% RSLogix 500 project WN16_175291_P_WFI_01_1.RSS, saved by version 8.10.00.24 %
PROJECT "RX72EPIS"    % processor: SLC 500, 1747-L541 %

PROGRAM FILES
  LAD 2   11 rungs
  LAD 3 "table_entr"  31 rungs
  LAD 4 "consigne"  87 rungs
  LAD 5 "communicat"  10 rungs
  LAD 6 "alarmes"  55 rungs
  LAD 7 "programme"  27 rungs
  LAD 8 "pid"  41 rungs
  LAD 9 "affichage"  22 rungs
  LAD 10 "table_sort"  54 rungs
  LAD 29 "IN_TOC"  9 rungs  % TABLE ENTREE/ SOUS-ROUTINE TOC %
  LAD 30 "TOC"  25 rungs  % SOUS-ROUTINE TOC %

DATA FILES
  O0 OUTPUT  6 elements
  I1 INPUT  8 elements
  S2 STATUS  164 elements
  B3 BINARY  18 elements
  T4 TIMER  61 elements
  C5 COUNTER  6 elements
  R6 CONTROL  1 elements
  N7 INTEGER  11 elements
  F8 FLOAT  11 elements
  B9   21 elements
  B10   21 elements
  N11   75 elements
  N12   11 elements
  N13   12 elements
  N14   11 elements
  N15   11 elements
  N16   6 elements
  N17   2 elements
  B18   4 elements
  N19   98 elements
  T20   25 elements
  B21   7 elements
  N24   75 elements
  N25   31 elements
  N27   56 elements
  N28   26 elements
  N30 TOC  30 elements  % Data Files/ Analyseur TOC %
  T31 TOC TIMER  10 elements  % Data Files/ Analyseur TOC %

LADDER 2
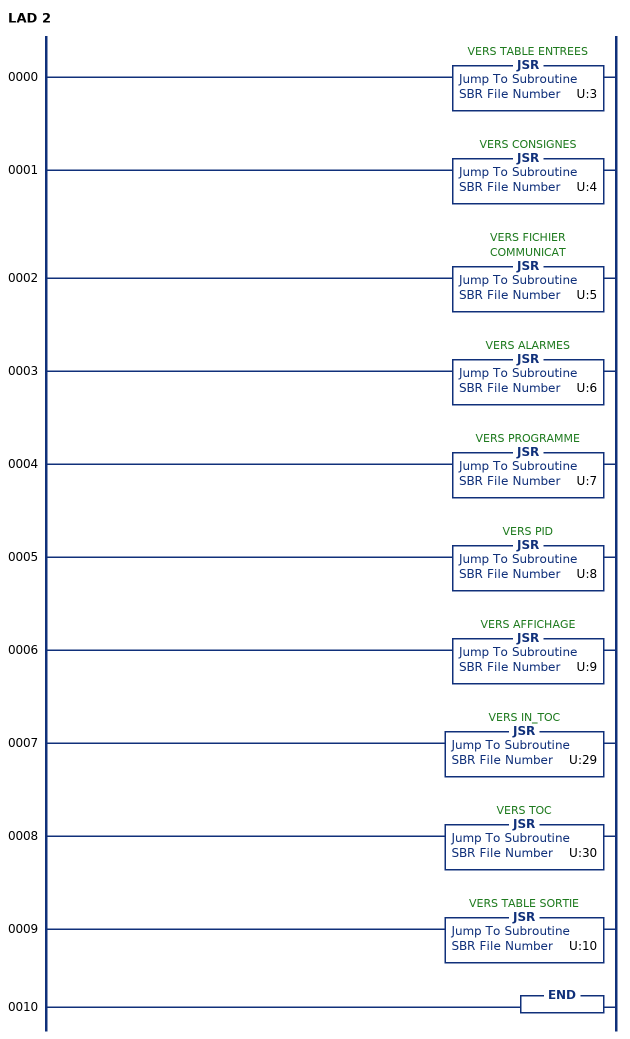
% Rung: 0 %
SOR JSR U:3 EOR
%   U:3  "VERS TABLE ENTREES" %
% Rung: 1 %
SOR JSR U:4 EOR
%   U:4  "VERS CONSIGNES" %
% Rung: 2 %
SOR JSR U:5 EOR
%   U:5  "VERS FICHIER COMMUNICAT" %
% Rung: 3 %
SOR JSR U:6 EOR
%   U:6  "VERS ALARMES" %
% Rung: 4 %
SOR JSR U:7 EOR
%   U:7  "VERS PROGRAMME" %
% Rung: 5 %
SOR JSR U:8 EOR
%   U:8  "VERS PID" %
% Rung: 6 %
SOR JSR U:9 EOR
%   U:9  "VERS AFFICHAGE" %
% Rung: 7 %
SOR JSR U:29 EOR
%   U:29  "VERS IN_TOC" %
% Rung: 8 %
SOR JSR U:30 EOR
%   U:30  "VERS TOC" %
% Rung: 9 %
SOR JSR U:10 EOR
%   U:10  "VERS TABLE SORTIE" %
% Rung: 10 %
SOR END EOR

LADDER 3 "table_entr"
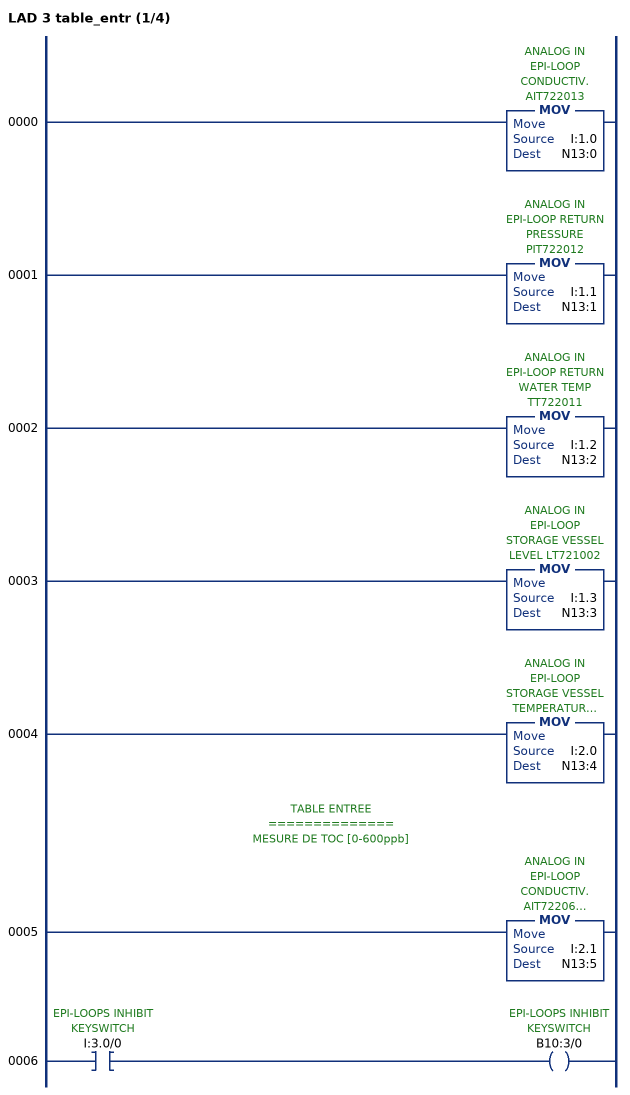
% Rung: 0 %
SOR MOV I:1.0 N13:0 EOR
%   N13:0  "ANALOG IN EPI-LOOP CONDUCTIV. AIT722013" %
% Rung: 1 %
SOR MOV I:1.1 N13:1 EOR
%   N13:1  "ANALOG IN EPI-LOOP RETURN PRESSURE PIT722012" %
% Rung: 2 %
SOR MOV I:1.2 N13:2 EOR
%   N13:2  "ANALOG IN EPI-LOOP RETURN WATER TEMP TT722011" %
% Rung: 3 %
SOR MOV I:1.3 N13:3 EOR
%   N13:3  "ANALOG IN EPI-LOOP STORAGE VESSEL LEVEL LT721002" %
% Rung: 4 %
SOR MOV I:2.0 N13:4 EOR
%   N13:4  "ANALOG IN EPI-LOOP STORAGE VESSEL TEMPERATURE TT721005" %
% Rung: 5 %
% TABLE ENTREE
% ==============
% MESURE DE TOC [0-600ppb] %
SOR MOV I:2.1 N13:5 EOR
%   N13:5  AT_M3  "ANALOG IN EPI-LOOP CONDUCTIV. AIT722062" %
% Rung: 6 %
SOR XIC I:3.0/0 OTE B10:3/0 EOR
%   I:3.0/0  "EPI-LOOPS INHIBIT KEYSWITCH" %
%   B10:3/0  "EPI-LOOPS INHIBIT KEYSWITCH" %

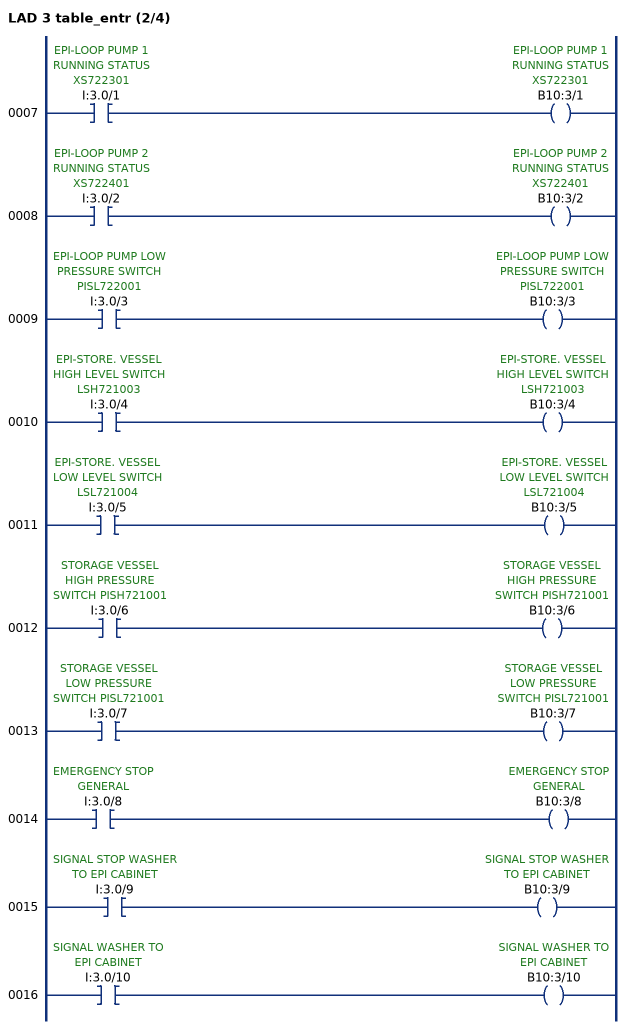
% Rung: 7 %
SOR XIC I:3.0/1 OTE B10:3/1 EOR
%   I:3.0/1  "EPI-LOOP PUMP 1 RUNNING STATUS XS722301" %
%   B10:3/1  "EPI-LOOP PUMP 1 RUNNING STATUS XS722301" %
% Rung: 8 %
SOR XIC I:3.0/2 OTE B10:3/2 EOR
%   I:3.0/2  "EPI-LOOP PUMP 2 RUNNING STATUS XS722401" %
%   B10:3/2  "EPI-LOOP PUMP 2 RUNNING STATUS XS722401" %
% Rung: 9 %
SOR XIC I:3.0/3 OTE B10:3/3 EOR
%   I:3.0/3  "EPI-LOOP PUMP LOW PRESSURE SWITCH PISL722001" %
%   B10:3/3  "EPI-LOOP PUMP LOW PRESSURE SWITCH PISL722001" %
% Rung: 10 %
SOR XIC I:3.0/4 OTE B10:3/4 EOR
%   I:3.0/4  "EPI-STORE. VESSEL HIGH LEVEL SWITCH LSH721003" %
%   B10:3/4  "EPI-STORE. VESSEL HIGH LEVEL SWITCH LSH721003" %
% Rung: 11 %
SOR XIC I:3.0/5 OTE B10:3/5 EOR
%   I:3.0/5  "EPI-STORE. VESSEL LOW LEVEL SWITCH LSL721004" %
%   B10:3/5  "EPI-STORE. VESSEL LOW LEVEL SWITCH LSL721004" %
% Rung: 12 %
SOR XIC I:3.0/6 OTE B10:3/6 EOR
%   I:3.0/6  "STORAGE VESSEL HIGH PRESSURE SWITCH PISH721001" %
%   B10:3/6  "STORAGE VESSEL HIGH PRESSURE SWITCH PISH721001" %
% Rung: 13 %
SOR XIC I:3.0/7 OTE B10:3/7 EOR
%   I:3.0/7  "STORAGE VESSEL LOW PRESSURE SWITCH PISL721001" %
%   B10:3/7  "STORAGE VESSEL LOW PRESSURE SWITCH PISL721001" %
% Rung: 14 %
SOR XIC I:3.0/8 OTE B10:3/8 EOR
%   I:3.0/8  "EMERGENCY STOP GENERAL" %
%   B10:3/8  "EMERGENCY STOP GENERAL" %
% Rung: 15 %
SOR XIC I:3.0/9 OTE B10:3/9 EOR
%   I:3.0/9  "SIGNAL STOP WASHER TO EPI CABINET" %
%   B10:3/9  "SIGNAL STOP WASHER TO EPI CABINET" %
% Rung: 16 %
SOR XIC I:3.0/10 OTE B10:3/10 EOR
%   I:3.0/10  "SIGNAL WASHER TO EPI CABINET" %
%   B10:3/10  "SIGNAL WASHER TO EPI CABINET" %

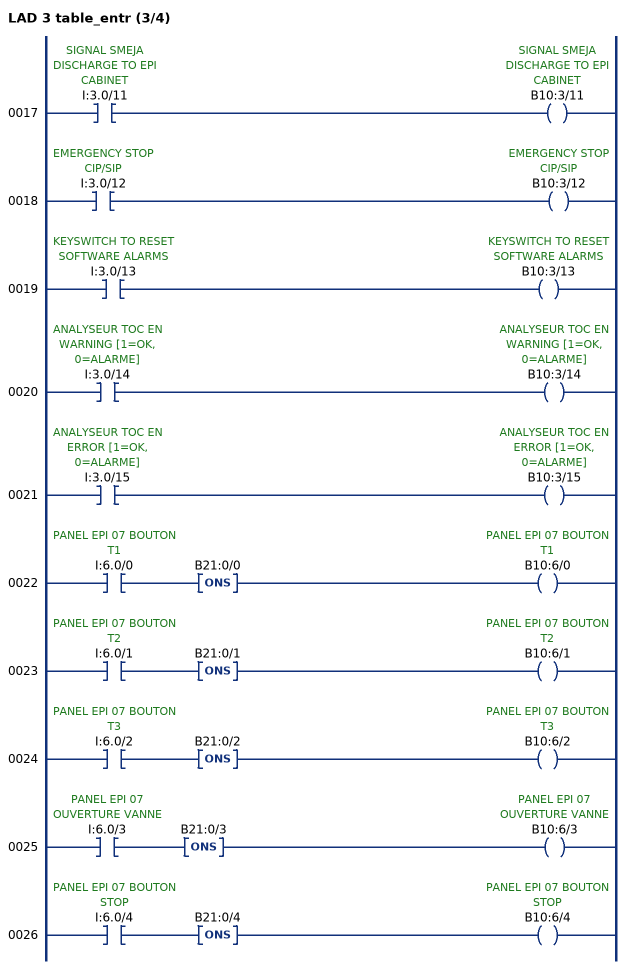
% Rung: 17 %
SOR XIC I:3.0/11 OTE B10:3/11 EOR
%   I:3.0/11  "SIGNAL SMEJA DISCHARGE TO EPI CABINET" %
%   B10:3/11  "SIGNAL SMEJA DISCHARGE TO EPI CABINET" %
% Rung: 18 %
SOR XIC I:3.0/12 OTE B10:3/12 EOR
%   I:3.0/12  "EMERGENCY STOP CIP/SIP" %
%   B10:3/12  "EMERGENCY STOP CIP/SIP" %
% Rung: 19 %
SOR XIC I:3.0/13 OTE B10:3/13 EOR
%   I:3.0/13  "KEYSWITCH TO RESET SOFTWARE ALARMS" %
%   B10:3/13  "KEYSWITCH TO RESET SOFTWARE ALARMS" %
% Rung: 20 %
SOR XIC I:3.0/14 OTE B10:3/14 EOR
%   I:3.0/14  "ANALYSEUR TOC EN WARNING [1=OK, 0=ALARME]" %
%   B10:3/14  "ANALYSEUR TOC EN WARNING [1=OK, 0=ALARME]" %
% Rung: 21 %
SOR XIC I:3.0/15 OTE B10:3/15 EOR
%   I:3.0/15  "ANALYSEUR TOC EN ERROR [1=OK, 0=ALARME]" %
%   B10:3/15  "ANALYSEUR TOC EN ERROR [1=OK, 0=ALARME]" %
% Rung: 22 %
SOR XIC I:6.0/0 OSR B21:0/0 OTE B10:6/0 EOR
%   I:6.0/0  "PANEL EPI 07 BOUTON T1" %
%   B10:6/0  "PANEL EPI 07 BOUTON T1" %
% Rung: 23 %
SOR XIC I:6.0/1 OSR B21:0/1 OTE B10:6/1 EOR
%   I:6.0/1  "PANEL EPI 07 BOUTON T2" %
%   B10:6/1  "PANEL EPI 07 BOUTON T2" %
% Rung: 24 %
SOR XIC I:6.0/2 OSR B21:0/2 OTE B10:6/2 EOR
%   I:6.0/2  "PANEL EPI 07 BOUTON T3" %
%   B10:6/2  "PANEL EPI 07 BOUTON T3" %
% Rung: 25 %
SOR XIC I:6.0/3 OSR B21:0/3 OTE B10:6/3 EOR
%   I:6.0/3  "PANEL EPI 07 OUVERTURE VANNE" %
%   B10:6/3  "PANEL EPI 07 OUVERTURE VANNE" %
% Rung: 26 %
SOR XIC I:6.0/4 OSR B21:0/4 OTE B10:6/4 EOR
%   I:6.0/4  "PANEL EPI 07 BOUTON STOP" %
%   B10:6/4  "PANEL EPI 07 BOUTON STOP" %

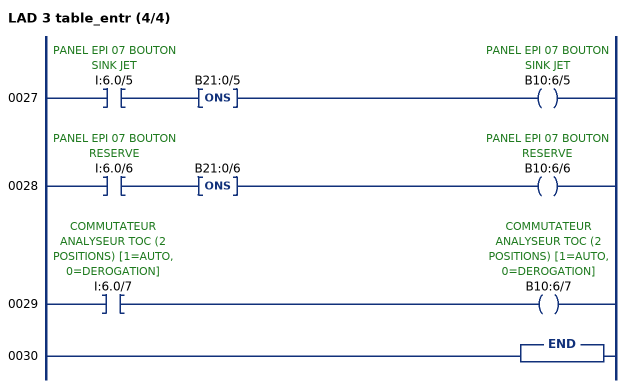
% Rung: 27 %
SOR XIC I:6.0/5 OSR B21:0/5 OTE B10:6/5 EOR
%   I:6.0/5  "PANEL EPI 07 BOUTON SINK JET" %
%   B10:6/5  "PANEL EPI 07 BOUTON SINK JET" %
% Rung: 28 %
SOR XIC I:6.0/6 OSR B21:0/6 OTE B10:6/6 EOR
%   I:6.0/6  "PANEL EPI 07 BOUTON RESERVE" %
%   B10:6/6  "PANEL EPI 07 BOUTON RESERVE" %
% Rung: 29 %
SOR XIC I:6.0/7 OTE B10:6/7 EOR
%   I:6.0/7  "COMMUTATEUR ANALYSEUR TOC (2 POSITIONS) [1=AUTO, 0=DEROGATION]" %
%   B10:6/7  "COMMUTATEUR ANALYSEUR TOC (2 POSITIONS) [1=AUTO, 0=DEROGATION]" %
% Rung: 30 %
SOR END EOR

LADDER 4 "consigne"
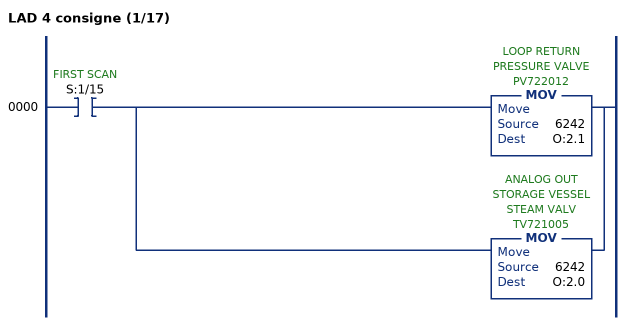
% Rung: 0 %
SOR XIC S:1/15 BST MOV 6242 O:2.1 NXB MOV 6242 O:2.0 BND EOR
%   S:1/15  "FIRST SCAN" %
%   O:2.1  "LOOP RETURN PRESSURE VALVE PV722012" %
%   O:2.0  "ANALOG OUT STORAGE VESSEL STEAM VALV TV721005" %

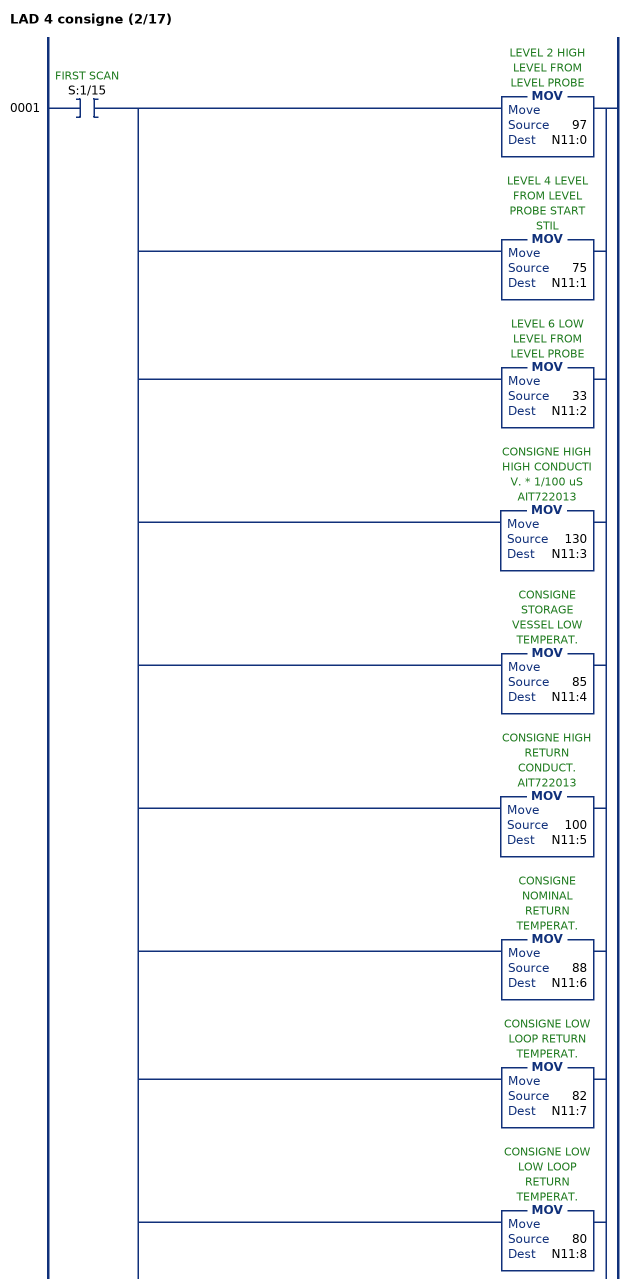

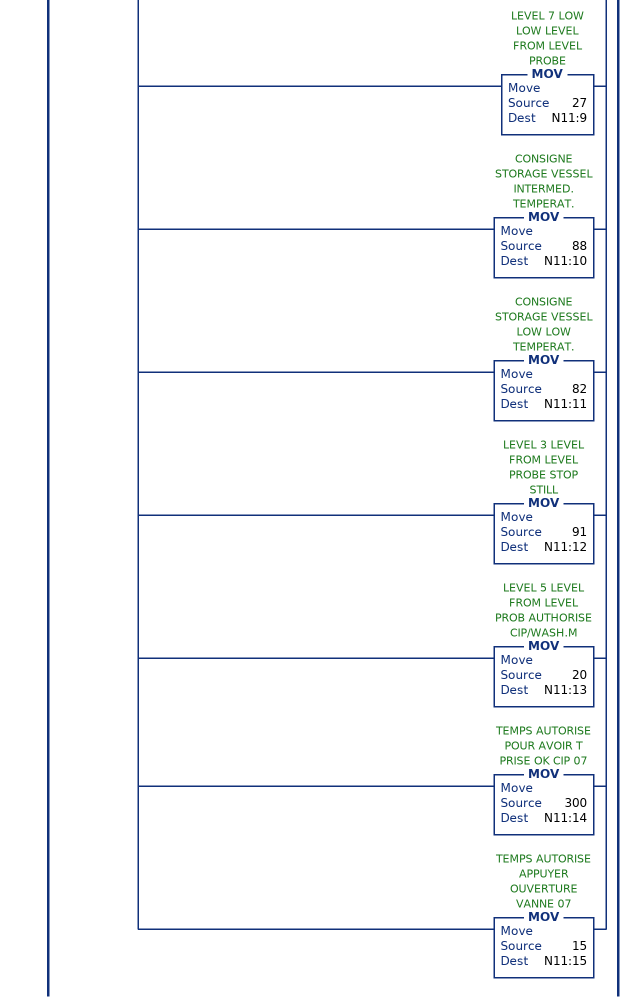
% Rung: 1 %
SOR XIC S:1/15 BST MOV 97 N11:0 NXB MOV 75 N11:1 NXB MOV 33 N11:2 NXB MOV 130 N11:3 NXB MOV 85 N11:4 NXB MOV 100 N11:5 NXB MOV 88 N11:6 NXB MOV 82 N11:7 NXB MOV 80 N11:8 NXB MOV 27 N11:9 NXB MOV 88 N11:10 NXB MOV 82 N11:11 NXB MOV 91 N11:12 NXB MOV 20 N11:13 NXB MOV 300 N11:14 NXB MOV 15 N11:15 BND EOR
%   S:1/15  "FIRST SCAN" %
%   N11:0  "LEVEL 2 HIGH LEVEL FROM LEVEL PROBE" %
%   N11:1  "LEVEL 4 LEVEL FROM LEVEL PROBE START STIL" %
%   N11:2  "LEVEL 6 LOW LEVEL FROM LEVEL PROBE" %
%   N11:3  "CONSIGNE HIGH HIGH CONDUCTIV. * 1/100 uS AIT722013" %
%   N11:4  "CONSIGNE STORAGE VESSEL LOW TEMPERAT." %
%   N11:5  "CONSIGNE HIGH RETURN CONDUCT. AIT722013" %
%   N11:6  "CONSIGNE NOMINAL RETURN TEMPERAT." %
%   N11:7  "CONSIGNE LOW LOOP RETURN TEMPERAT." %
%   N11:8  "CONSIGNE LOW LOW LOOP RETURN TEMPERAT." %
%   N11:9  "LEVEL 7 LOW LOW LEVEL FROM LEVEL PROBE" %
%   N11:10  "CONSIGNE STORAGE VESSEL INTERMED. TEMPERAT." %
%   N11:11  "CONSIGNE STORAGE VESSEL LOW LOW TEMPERAT." %
%   N11:12  "LEVEL 3 LEVEL FROM LEVEL PROBE STOP STILL" %
%   N11:13  "LEVEL 5 LEVEL FROM LEVEL PROB AUTHORISE CIP/WASH.M" %
%   N11:14  "TEMPS AUTORISE POUR AVOIR T PRISE OK CIP 07" %
%   N11:15  "TEMPS AUTORISE APPUYER OUVERTURE VANNE 07" %

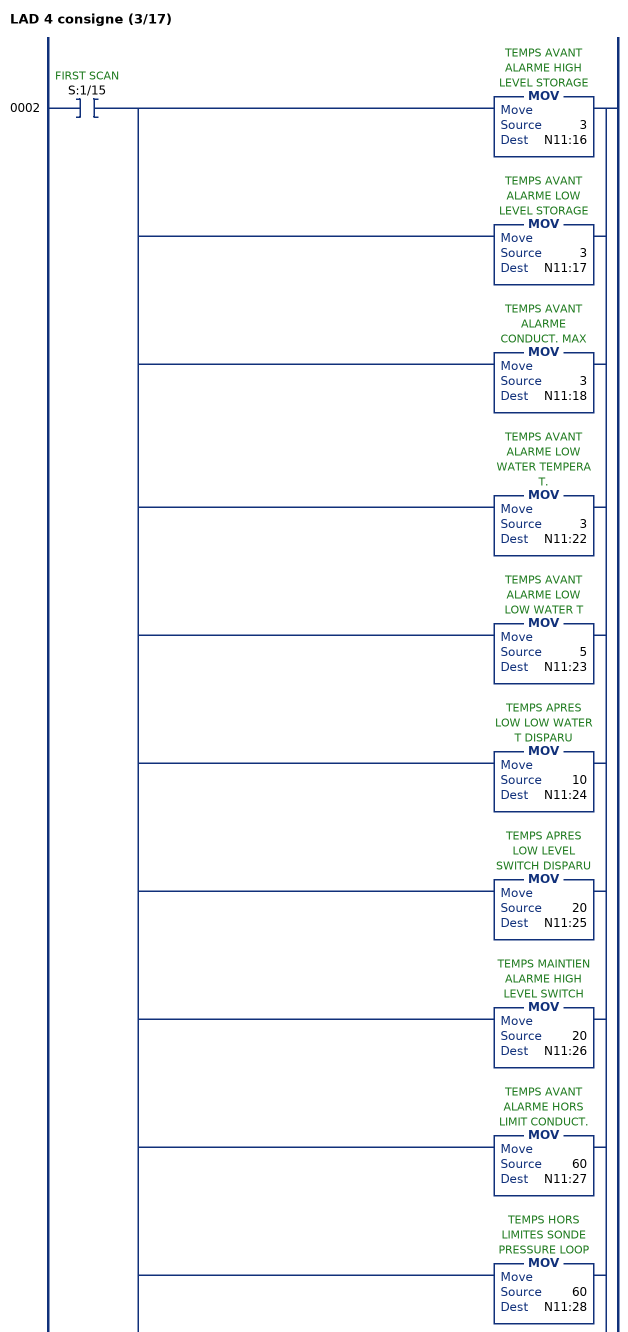

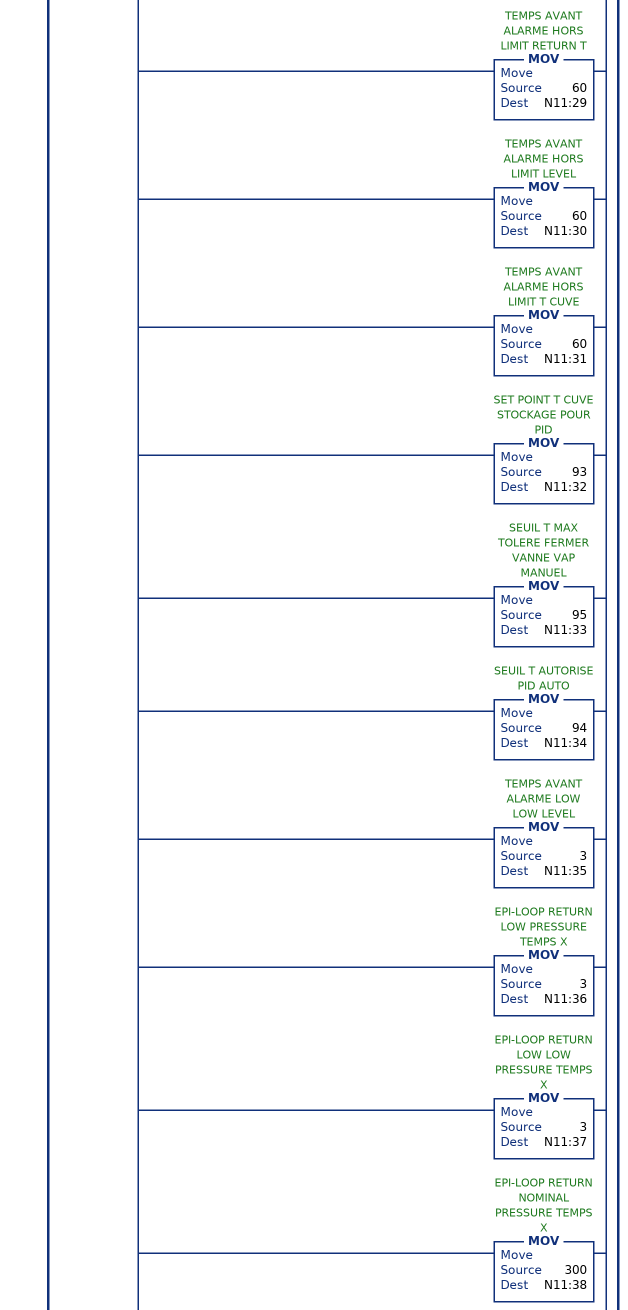

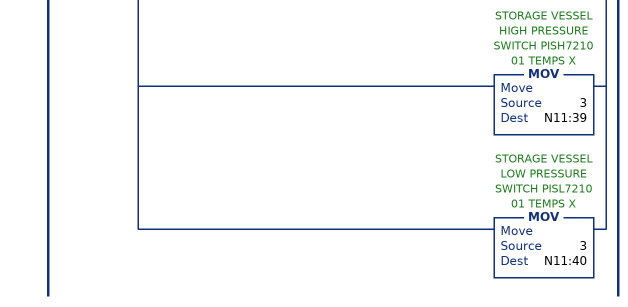
% Rung: 2 %
SOR XIC S:1/15 BST MOV 3 N11:16 NXB MOV 3 N11:17 NXB MOV 3 N11:18 NXB MOV 3 N11:22 NXB MOV 5 N11:23 NXB MOV 10 N11:24 NXB MOV 20 N11:25 NXB MOV 20 N11:26 NXB MOV 60 N11:27 NXB MOV 60 N11:28 NXB MOV 60 N11:29 NXB MOV 60 N11:30 NXB MOV 60 N11:31 NXB MOV 93 N11:32 NXB MOV 95 N11:33 NXB MOV 94 N11:34 NXB MOV 3 N11:35 NXB MOV 3 N11:36 NXB MOV 3 N11:37 NXB MOV 300 N11:38 NXB MOV 3 N11:39 NXB MOV 3 N11:40 BND EOR
%   S:1/15  "FIRST SCAN" %
%   N11:16  "TEMPS AVANT ALARME HIGH LEVEL STORAGE" %
%   N11:17  "TEMPS AVANT ALARME LOW LEVEL STORAGE" %
%   N11:18  "TEMPS AVANT ALARME CONDUCT. MAX" %
%   N11:22  "TEMPS AVANT ALARME LOW WATER TEMPERAT." %
%   N11:23  "TEMPS AVANT ALARME LOW LOW WATER T" %
%   N11:24  "TEMPS APRES LOW LOW WATER T DISPARU" %
%   N11:25  "TEMPS APRES LOW LEVEL SWITCH DISPARU" %
%   N11:26  "TEMPS MAINTIEN ALARME HIGH LEVEL SWITCH" %
%   N11:27  "TEMPS AVANT ALARME HORS LIMIT CONDUCT." %
%   N11:28  "TEMPS HORS LIMITES SONDE PRESSURE LOOP" %
%   N11:29  "TEMPS AVANT ALARME HORS LIMIT RETURN T" %
%   N11:30  "TEMPS AVANT ALARME HORS LIMIT LEVEL" %
%   N11:31  "TEMPS AVANT ALARME HORS LIMIT T CUVE" %
%   N11:32  "SET POINT T CUVE STOCKAGE POUR PID" %
%   N11:33  "SEUIL T MAX TOLERE FERMER VANNE VAP MANUEL" %
%   N11:34  "SEUIL T AUTORISE PID AUTO" %
%   N11:35  "TEMPS AVANT ALARME LOW LOW LEVEL" %
%   N11:36  "EPI-LOOP RETURN LOW PRESSURE TEMPS X" %
%   N11:37  "EPI-LOOP RETURN LOW LOW PRESSURE TEMPS X" %
%   N11:38  "EPI-LOOP RETURN NOMINAL PRESSURE TEMPS X" %
%   N11:39  "STORAGE VESSEL HIGH PRESSURE SWITCH PISH721001 TEMPS X" %
%   N11:40  "STORAGE VESSEL LOW PRESSURE SWITCH PISL721001 TEMPS X" %

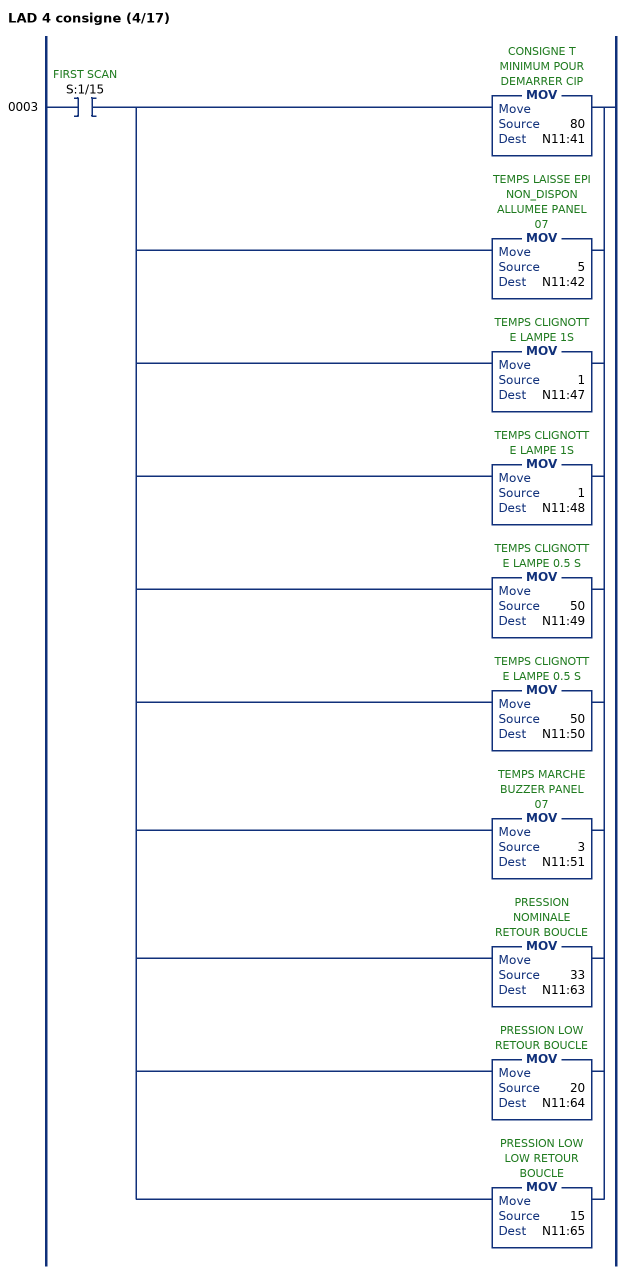
% Rung: 3 %
SOR XIC S:1/15 BST MOV 80 N11:41 NXB MOV 5 N11:42 NXB MOV 1 N11:47 NXB MOV 1 N11:48 NXB MOV 50 N11:49 NXB MOV 50 N11:50 NXB MOV 3 N11:51 NXB MOV 33 N11:63 NXB MOV 20 N11:64 NXB MOV 15 N11:65 BND EOR
%   S:1/15  "FIRST SCAN" %
%   N11:41  "CONSIGNE T MINIMUM POUR DEMARRER CIP" %
%   N11:42  "TEMPS LAISSE EPI NON_DISPON ALLUMEE PANEL 07" %
%   N11:47  "TEMPS CLIGNOTTE LAMPE 1S" %
%   N11:48  "TEMPS CLIGNOTTE LAMPE 1S" %
%   N11:49  "TEMPS CLIGNOTTE LAMPE 0.5 S" %
%   N11:50  "TEMPS CLIGNOTTE LAMPE 0.5 S" %
%   N11:51  "TEMPS MARCHE BUZZER PANEL 07" %
%   N11:63  "PRESSION NOMINALE RETOUR BOUCLE" %
%   N11:64  "PRESSION LOW RETOUR BOUCLE" %
%   N11:65  "PRESSION LOW LOW RETOUR BOUCLE" %

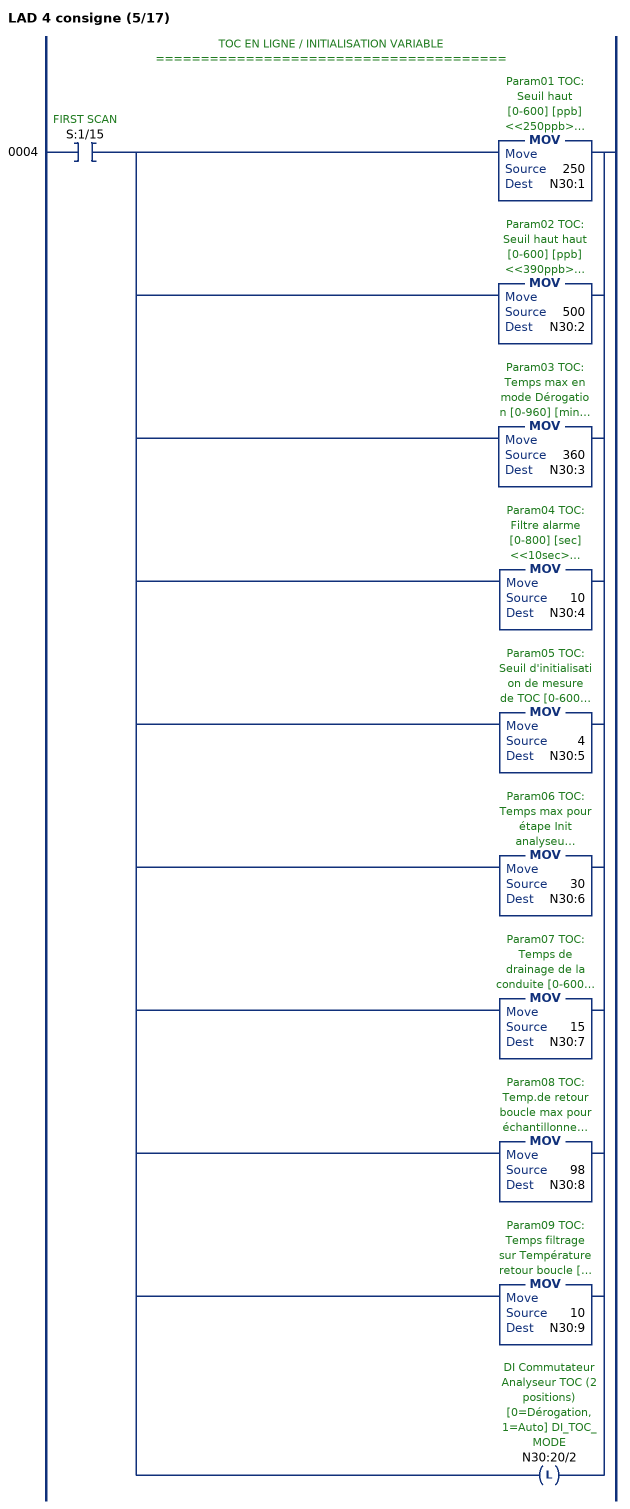
% Rung: 4 %
% TOC EN LIGNE / INITIALISATION VARIABLE
% ======================================= %
SOR XIC S:1/15 BST MOV 250 N30:1 NXB MOV 500 N30:2 NXB MOV 360 N30:3 NXB MOV 10 N30:4 NXB MOV 4 N30:5 NXB MOV 30 N30:6 NXB MOV 15 N30:7 NXB MOV 98 N30:8 NXB MOV 10 N30:9 NXB OTL N30:20/2 BND EOR
%   S:1/15  "FIRST SCAN" %
%   N30:1  AI_AT_M3_LIMH  "Param01 TOC: Seuil haut [0-600] [ppb] <<250ppb>>" %
%   N30:2  AI_AT_M3_LIMHH  "Param02 TOC: Seuil haut haut [0-600] [ppb] <<390ppb>>" %
%   N30:3  AI_TOC_DEROG_LIMH  "Param03 TOC: Temps max en mode Dérogation [0-960] [min] <<360min>>" %
%   N30:4  AI_AT_M3_ALM_HH_DL  "Param04 TOC: Filtre alarme [0-800] [sec] <<10sec>>" %
%   N30:5  AI_AT_M3_MIN  "Param05 TOC: Seuil d'initialisation de mesure de TOC [0-600] [ppb] <<4ppb>>" %
%   N30:6  AI_TOC_INIT_LIMH  "Param06 TOC: Temps max pour étape Init analyseur [0-600] [min] <<30min>>" %
%   N30:7  AI_XV_M3_CMD_DELAY  "Param07 TOC: Temps de drainage de la conduite [0-600] [sec] <<15sec>>" %
%   N30:8  AI_TT_722011_LIMH  "Param08 TOC: Temp.de retour boucle max pour échantillonner [0-100] [°C] <<98°C>>" %
%   N30:9  AI_T_TT_722011_LIMH  "Param09 TOC: Temps filtrage sur Température retour boucle [] [min] <<10 min>>" %
%   N30:20/2  DI_TOC_MODE  "DI Commutateur Analyseur TOC (2 positions) [0=Dérogation, 1=Auto]" %

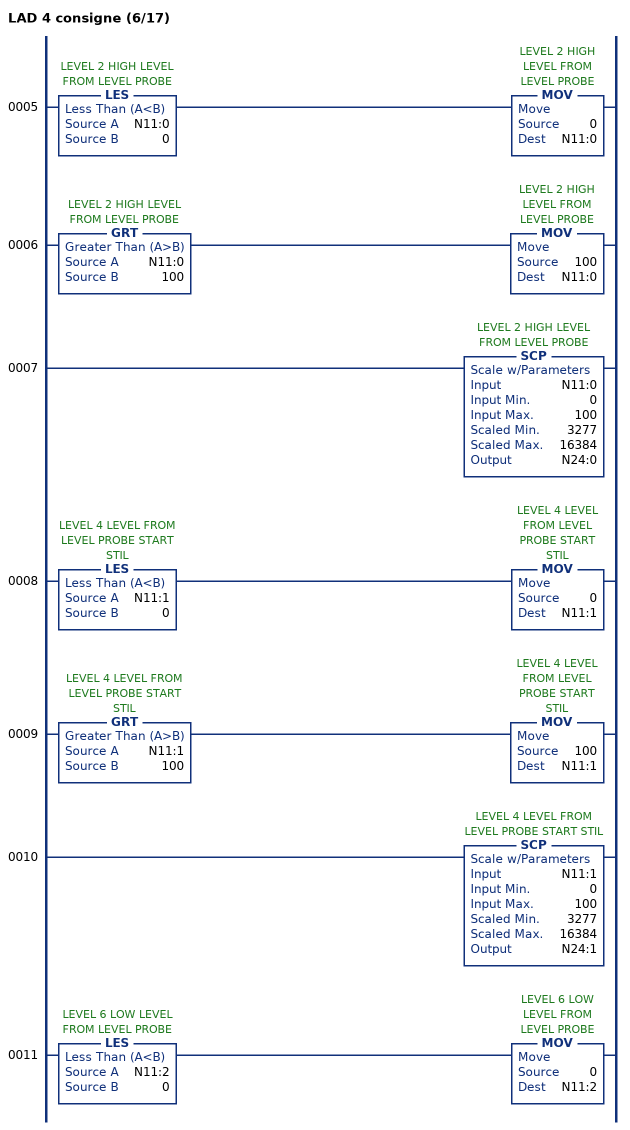
% Rung: 5 %
SOR LES N11:0 0 MOV 0 N11:0 EOR
%   N11:0  "LEVEL 2 HIGH LEVEL FROM LEVEL PROBE" %
% Rung: 6 %
SOR GRT N11:0 100 MOV 100 N11:0 EOR
%   N11:0  "LEVEL 2 HIGH LEVEL FROM LEVEL PROBE" %
% Rung: 7 %
SOR SCP N11:0 0 100 3277 16384 N24:0 EOR
%   N11:0  "LEVEL 2 HIGH LEVEL FROM LEVEL PROBE" %
%   N24:0  "LEVEL 2 HIGH LEVEL FROM LEVEL PROBE" %
% Rung: 8 %
SOR LES N11:1 0 MOV 0 N11:1 EOR
%   N11:1  "LEVEL 4 LEVEL FROM LEVEL PROBE START STIL" %
% Rung: 9 %
SOR GRT N11:1 100 MOV 100 N11:1 EOR
%   N11:1  "LEVEL 4 LEVEL FROM LEVEL PROBE START STIL" %
% Rung: 10 %
SOR SCP N11:1 0 100 3277 16384 N24:1 EOR
%   N11:1  "LEVEL 4 LEVEL FROM LEVEL PROBE START STIL" %
%   N24:1  "LEVEL 4 LEVEL FROM LEVEL PROBE START STIL" %
% Rung: 11 %
SOR LES N11:2 0 MOV 0 N11:2 EOR
%   N11:2  "LEVEL 6 LOW LEVEL FROM LEVEL PROBE" %

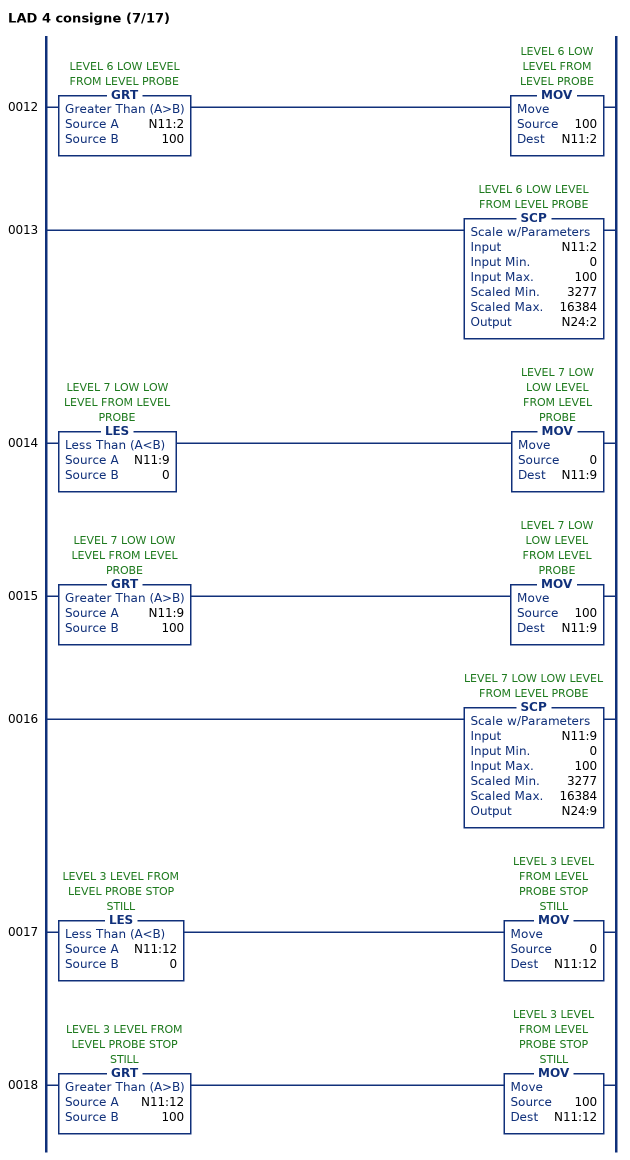
% Rung: 12 %
SOR GRT N11:2 100 MOV 100 N11:2 EOR
%   N11:2  "LEVEL 6 LOW LEVEL FROM LEVEL PROBE" %
% Rung: 13 %
SOR SCP N11:2 0 100 3277 16384 N24:2 EOR
%   N11:2  "LEVEL 6 LOW LEVEL FROM LEVEL PROBE" %
%   N24:2  "LEVEL 6 LOW LEVEL FROM LEVEL PROBE" %
% Rung: 14 %
SOR LES N11:9 0 MOV 0 N11:9 EOR
%   N11:9  "LEVEL 7 LOW LOW LEVEL FROM LEVEL PROBE" %
% Rung: 15 %
SOR GRT N11:9 100 MOV 100 N11:9 EOR
%   N11:9  "LEVEL 7 LOW LOW LEVEL FROM LEVEL PROBE" %
% Rung: 16 %
SOR SCP N11:9 0 100 3277 16384 N24:9 EOR
%   N11:9  "LEVEL 7 LOW LOW LEVEL FROM LEVEL PROBE" %
%   N24:9  "LEVEL 7 LOW LOW LEVEL FROM LEVEL PROBE" %
% Rung: 17 %
SOR LES N11:12 0 MOV 0 N11:12 EOR
%   N11:12  "LEVEL 3 LEVEL FROM LEVEL PROBE STOP STILL" %
% Rung: 18 %
SOR GRT N11:12 100 MOV 100 N11:12 EOR
%   N11:12  "LEVEL 3 LEVEL FROM LEVEL PROBE STOP STILL" %

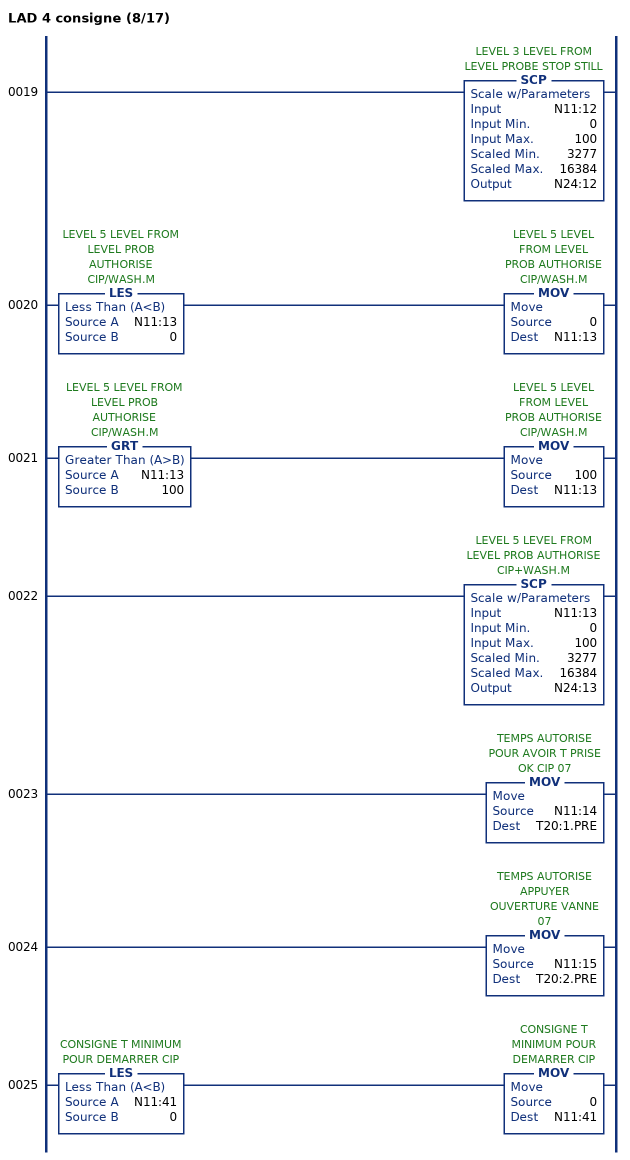
% Rung: 19 %
SOR SCP N11:12 0 100 3277 16384 N24:12 EOR
%   N11:12  "LEVEL 3 LEVEL FROM LEVEL PROBE STOP STILL" %
%   N24:12  "LEVEL 3 LEVEL FROM LEVEL PROBE STOP STILL" %
% Rung: 20 %
SOR LES N11:13 0 MOV 0 N11:13 EOR
%   N11:13  "LEVEL 5 LEVEL FROM LEVEL PROB AUTHORISE CIP/WASH.M" %
% Rung: 21 %
SOR GRT N11:13 100 MOV 100 N11:13 EOR
%   N11:13  "LEVEL 5 LEVEL FROM LEVEL PROB AUTHORISE CIP/WASH.M" %
% Rung: 22 %
SOR SCP N11:13 0 100 3277 16384 N24:13 EOR
%   N11:13  "LEVEL 5 LEVEL FROM LEVEL PROB AUTHORISE CIP/WASH.M" %
%   N24:13  "LEVEL 5 LEVEL FROM LEVEL PROB AUTHORISE CIP+WASH.M" %
% Rung: 23 %
SOR MOV N11:14 T20:1.PRE EOR
%   N11:14  "TEMPS AUTORISE POUR AVOIR T PRISE OK CIP 07" %
%   T20:1.PRE  "TEMPS AUTORISE POUR AVOIR T PRISE OK CIP 07" %
% Rung: 24 %
SOR MOV N11:15 T20:2.PRE EOR
%   N11:15  "TEMPS AUTORISE APPUYER OUVERTURE VANNE 07" %
%   T20:2.PRE  "TEMPS AUTORISE APPUYER OUVERTURE VANNE 07" %
% Rung: 25 %
SOR LES N11:41 0 MOV 0 N11:41 EOR
%   N11:41  "CONSIGNE T MINIMUM POUR DEMARRER CIP" %

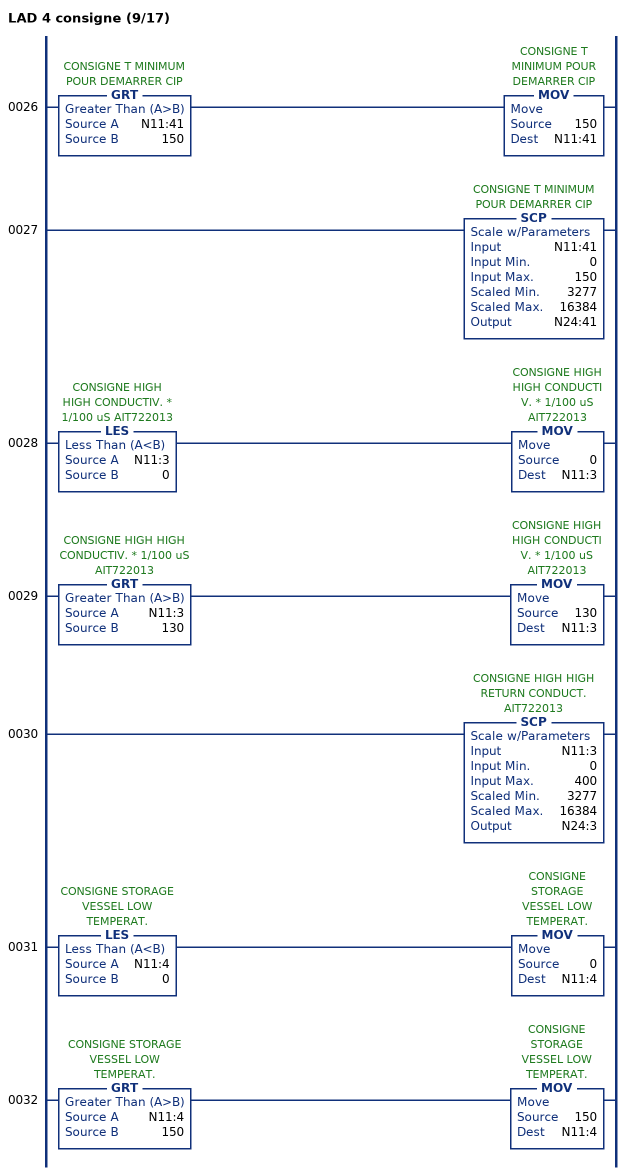
% Rung: 26 %
SOR GRT N11:41 150 MOV 150 N11:41 EOR
%   N11:41  "CONSIGNE T MINIMUM POUR DEMARRER CIP" %
% Rung: 27 %
SOR SCP N11:41 0 150 3277 16384 N24:41 EOR
%   N11:41  "CONSIGNE T MINIMUM POUR DEMARRER CIP" %
%   N24:41  "CONSIGNE T MINIMUM POUR DEMARRER CIP" %
% Rung: 28 %
SOR LES N11:3 0 MOV 0 N11:3 EOR
%   N11:3  "CONSIGNE HIGH HIGH CONDUCTIV. * 1/100 uS AIT722013" %
% Rung: 29 %
SOR GRT N11:3 130 MOV 130 N11:3 EOR
%   N11:3  "CONSIGNE HIGH HIGH CONDUCTIV. * 1/100 uS AIT722013" %
% Rung: 30 %
SOR SCP N11:3 0 400 3277 16384 N24:3 EOR
%   N11:3  "CONSIGNE HIGH HIGH CONDUCTIV. * 1/100 uS AIT722013" %
%   N24:3  "CONSIGNE HIGH HIGH RETURN CONDUCT. AIT722013" %
% Rung: 31 %
SOR LES N11:4 0 MOV 0 N11:4 EOR
%   N11:4  "CONSIGNE STORAGE VESSEL LOW TEMPERAT." %
% Rung: 32 %
SOR GRT N11:4 150 MOV 150 N11:4 EOR
%   N11:4  "CONSIGNE STORAGE VESSEL LOW TEMPERAT." %

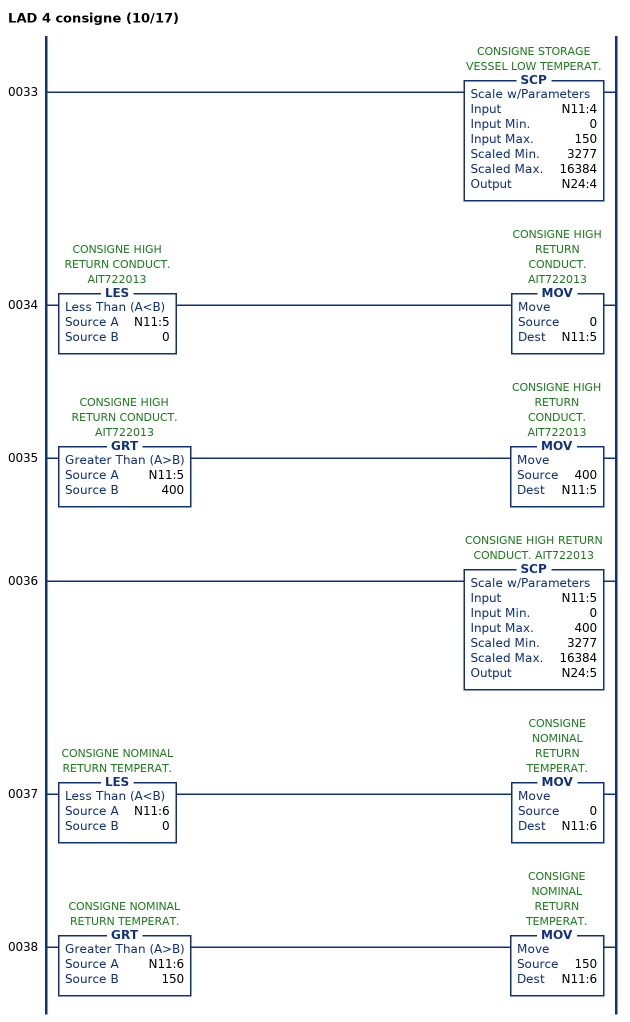
% Rung: 33 %
SOR SCP N11:4 0 150 3277 16384 N24:4 EOR
%   N11:4  "CONSIGNE STORAGE VESSEL LOW TEMPERAT." %
%   N24:4  "CONSIGNE STORAGE VESSEL LOW TEMPERAT." %
% Rung: 34 %
SOR LES N11:5 0 MOV 0 N11:5 EOR
%   N11:5  "CONSIGNE HIGH RETURN CONDUCT. AIT722013" %
% Rung: 35 %
SOR GRT N11:5 400 MOV 400 N11:5 EOR
%   N11:5  "CONSIGNE HIGH RETURN CONDUCT. AIT722013" %
% Rung: 36 %
SOR SCP N11:5 0 400 3277 16384 N24:5 EOR
%   N11:5  "CONSIGNE HIGH RETURN CONDUCT. AIT722013" %
%   N24:5  "CONSIGNE HIGH RETURN CONDUCT. AIT722013" %
% Rung: 37 %
SOR LES N11:6 0 MOV 0 N11:6 EOR
%   N11:6  "CONSIGNE NOMINAL RETURN TEMPERAT." %
% Rung: 38 %
SOR GRT N11:6 150 MOV 150 N11:6 EOR
%   N11:6  "CONSIGNE NOMINAL RETURN TEMPERAT." %

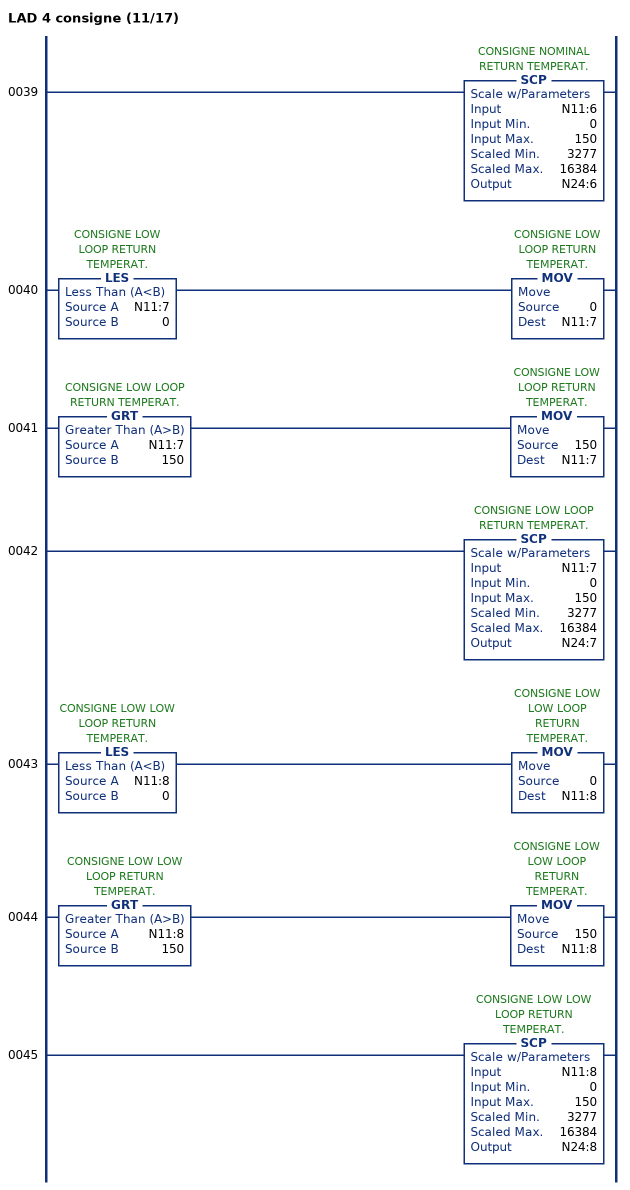
% Rung: 39 %
SOR SCP N11:6 0 150 3277 16384 N24:6 EOR
%   N11:6  "CONSIGNE NOMINAL RETURN TEMPERAT." %
%   N24:6  "CONSIGNE NOMINAL RETURN TEMPERAT." %
% Rung: 40 %
SOR LES N11:7 0 MOV 0 N11:7 EOR
%   N11:7  "CONSIGNE LOW LOOP RETURN TEMPERAT." %
% Rung: 41 %
SOR GRT N11:7 150 MOV 150 N11:7 EOR
%   N11:7  "CONSIGNE LOW LOOP RETURN TEMPERAT." %
% Rung: 42 %
SOR SCP N11:7 0 150 3277 16384 N24:7 EOR
%   N11:7  "CONSIGNE LOW LOOP RETURN TEMPERAT." %
%   N24:7  "CONSIGNE LOW LOOP RETURN TEMPERAT." %
% Rung: 43 %
SOR LES N11:8 0 MOV 0 N11:8 EOR
%   N11:8  "CONSIGNE LOW LOW LOOP RETURN TEMPERAT." %
% Rung: 44 %
SOR GRT N11:8 150 MOV 150 N11:8 EOR
%   N11:8  "CONSIGNE LOW LOW LOOP RETURN TEMPERAT." %
% Rung: 45 %
SOR SCP N11:8 0 150 3277 16384 N24:8 EOR
%   N11:8  "CONSIGNE LOW LOW LOOP RETURN TEMPERAT." %
%   N24:8  "CONSIGNE LOW LOW LOOP RETURN TEMPERAT." %

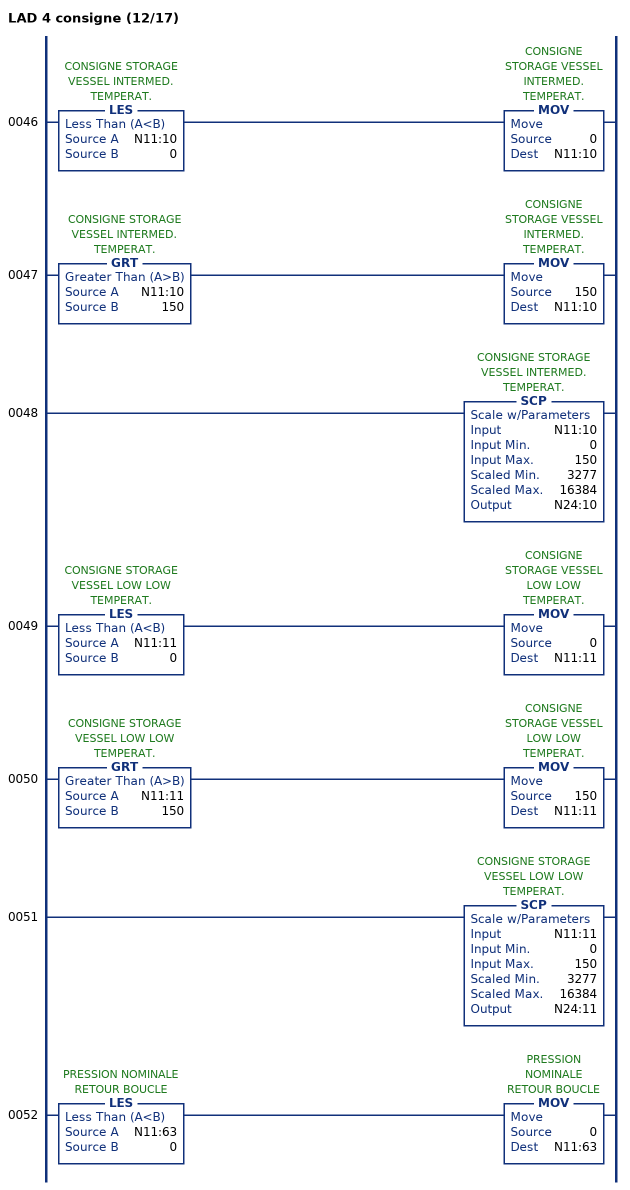
% Rung: 46 %
SOR LES N11:10 0 MOV 0 N11:10 EOR
%   N11:10  "CONSIGNE STORAGE VESSEL INTERMED. TEMPERAT." %
% Rung: 47 %
SOR GRT N11:10 150 MOV 150 N11:10 EOR
%   N11:10  "CONSIGNE STORAGE VESSEL INTERMED. TEMPERAT." %
% Rung: 48 %
SOR SCP N11:10 0 150 3277 16384 N24:10 EOR
%   N11:10  "CONSIGNE STORAGE VESSEL INTERMED. TEMPERAT." %
%   N24:10  "CONSIGNE STORAGE VESSEL INTERMED. TEMPERAT." %
% Rung: 49 %
SOR LES N11:11 0 MOV 0 N11:11 EOR
%   N11:11  "CONSIGNE STORAGE VESSEL LOW LOW TEMPERAT." %
% Rung: 50 %
SOR GRT N11:11 150 MOV 150 N11:11 EOR
%   N11:11  "CONSIGNE STORAGE VESSEL LOW LOW TEMPERAT." %
% Rung: 51 %
SOR SCP N11:11 0 150 3277 16384 N24:11 EOR
%   N11:11  "CONSIGNE STORAGE VESSEL LOW LOW TEMPERAT." %
%   N24:11  "CONSIGNE STORAGE VESSEL LOW LOW TEMPERAT." %
% Rung: 52 %
SOR LES N11:63 0 MOV 0 N11:63 EOR
%   N11:63  "PRESSION NOMINALE RETOUR BOUCLE" %

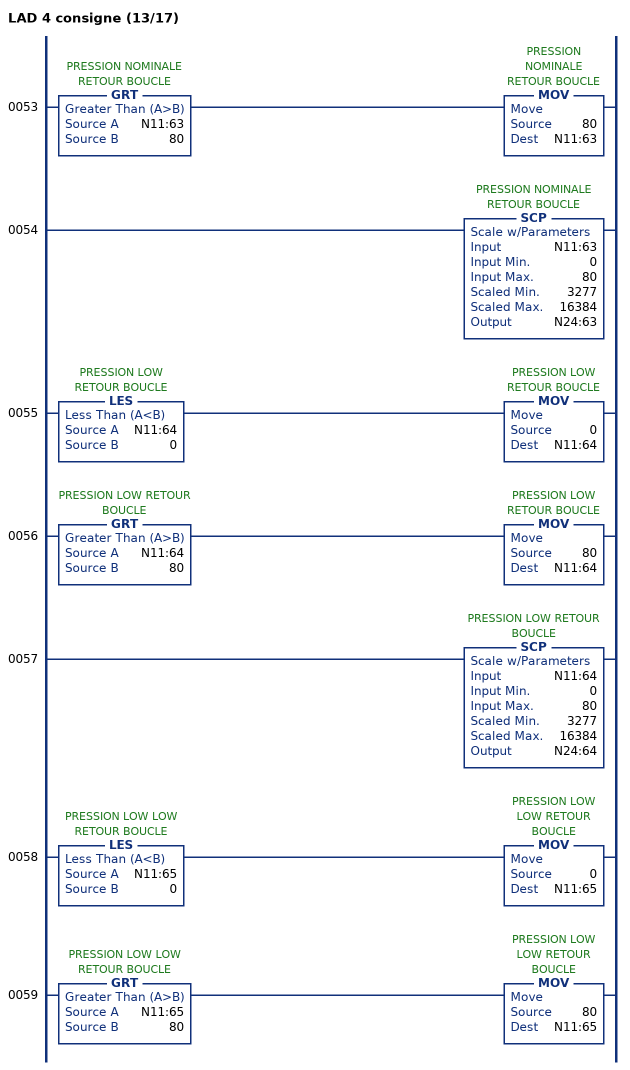
% Rung: 53 %
SOR GRT N11:63 80 MOV 80 N11:63 EOR
%   N11:63  "PRESSION NOMINALE RETOUR BOUCLE" %
% Rung: 54 %
SOR SCP N11:63 0 80 3277 16384 N24:63 EOR
%   N11:63  "PRESSION NOMINALE RETOUR BOUCLE" %
%   N24:63  "PRESSION NOMINALE RETOUR BOUCLE" %
% Rung: 55 %
SOR LES N11:64 0 MOV 0 N11:64 EOR
%   N11:64  "PRESSION LOW RETOUR BOUCLE" %
% Rung: 56 %
SOR GRT N11:64 80 MOV 80 N11:64 EOR
%   N11:64  "PRESSION LOW RETOUR BOUCLE" %
% Rung: 57 %
SOR SCP N11:64 0 80 3277 16384 N24:64 EOR
%   N11:64  "PRESSION LOW RETOUR BOUCLE" %
%   N24:64  "PRESSION LOW RETOUR BOUCLE" %
% Rung: 58 %
SOR LES N11:65 0 MOV 0 N11:65 EOR
%   N11:65  "PRESSION LOW LOW RETOUR BOUCLE" %
% Rung: 59 %
SOR GRT N11:65 80 MOV 80 N11:65 EOR
%   N11:65  "PRESSION LOW LOW RETOUR BOUCLE" %

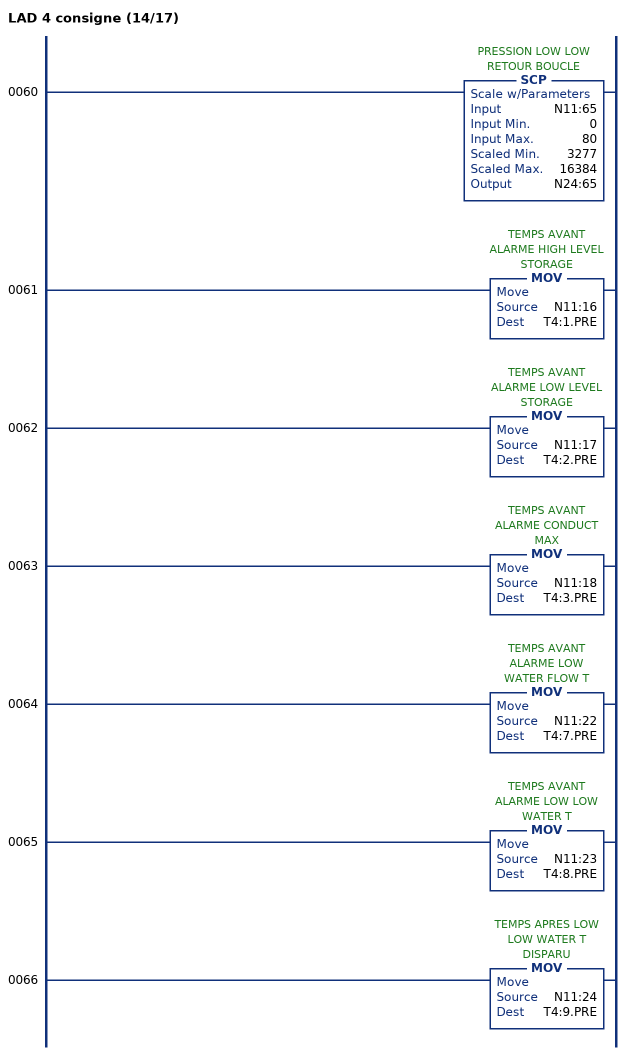
% Rung: 60 %
SOR SCP N11:65 0 80 3277 16384 N24:65 EOR
%   N11:65  "PRESSION LOW LOW RETOUR BOUCLE" %
%   N24:65  "PRESSION LOW LOW RETOUR BOUCLE" %
% Rung: 61 %
SOR MOV N11:16 T4:1.PRE EOR
%   N11:16  "TEMPS AVANT ALARME HIGH LEVEL STORAGE" %
%   T4:1.PRE  "TEMPS AVANT ALARME HIGH LEVEL STORAGE" %
% Rung: 62 %
SOR MOV N11:17 T4:2.PRE EOR
%   N11:17  "TEMPS AVANT ALARME LOW LEVEL STORAGE" %
%   T4:2.PRE  "TEMPS AVANT ALARME LOW LEVEL STORAGE" %
% Rung: 63 %
SOR MOV N11:18 T4:3.PRE EOR
%   N11:18  "TEMPS AVANT ALARME CONDUCT. MAX" %
%   T4:3.PRE  "TEMPS AVANT ALARME CONDUCT MAX" %
% Rung: 64 %
SOR MOV N11:22 T4:7.PRE EOR
%   N11:22  "TEMPS AVANT ALARME LOW WATER TEMPERAT." %
%   T4:7.PRE  "TEMPS AVANT ALARME LOW WATER FLOW T" %
% Rung: 65 %
SOR MOV N11:23 T4:8.PRE EOR
%   N11:23  "TEMPS AVANT ALARME LOW LOW WATER T" %
%   T4:8.PRE  "TEMPS AVANT ALARME LOW LOW WATER T" %
% Rung: 66 %
SOR MOV N11:24 T4:9.PRE EOR
%   N11:24  "TEMPS APRES LOW LOW WATER T DISPARU" %
%   T4:9.PRE  "TEMPS APRES LOW LOW WATER T DISPARU" %

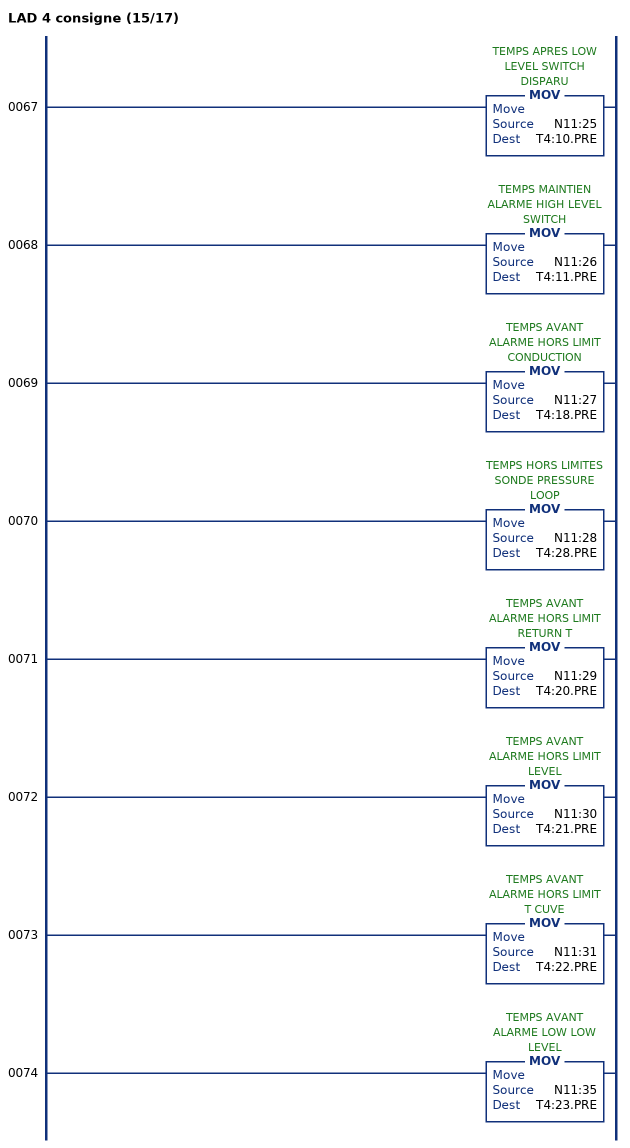
% Rung: 67 %
SOR MOV N11:25 T4:10.PRE EOR
%   N11:25  "TEMPS APRES LOW LEVEL SWITCH DISPARU" %
%   T4:10.PRE  "TEMPS APRES LOW LEVEL SWITCH DISPARU" %
% Rung: 68 %
SOR MOV N11:26 T4:11.PRE EOR
%   N11:26  "TEMPS MAINTIEN ALARME HIGH LEVEL SWITCH" %
%   T4:11.PRE  "TEMPS MAINTIEN ALARME HIGH LEVEL SWITCH" %
% Rung: 69 %
SOR MOV N11:27 T4:18.PRE EOR
%   N11:27  "TEMPS AVANT ALARME HORS LIMIT CONDUCT." %
%   T4:18.PRE  "TEMPS AVANT ALARME HORS LIMIT CONDUCTION" %
% Rung: 70 %
SOR MOV N11:28 T4:28.PRE EOR
%   N11:28  "TEMPS HORS LIMITES SONDE PRESSURE LOOP" %
%   T4:28.PRE  "TEMPS HORS LIMITES SONDE PRESSURE LOOP" %
% Rung: 71 %
SOR MOV N11:29 T4:20.PRE EOR
%   N11:29  "TEMPS AVANT ALARME HORS LIMIT RETURN T" %
%   T4:20.PRE  "TEMPS AVANT ALARME HORS LIMIT RETURN T" %
% Rung: 72 %
SOR MOV N11:30 T4:21.PRE EOR
%   N11:30  "TEMPS AVANT ALARME HORS LIMIT LEVEL" %
%   T4:21.PRE  "TEMPS AVANT ALARME HORS LIMIT LEVEL" %
% Rung: 73 %
SOR MOV N11:31 T4:22.PRE EOR
%   N11:31  "TEMPS AVANT ALARME HORS LIMIT T CUVE" %
%   T4:22.PRE  "TEMPS AVANT ALARME HORS LIMIT T CUVE" %
% Rung: 74 %
SOR MOV N11:35 T4:23.PRE EOR
%   N11:35  "TEMPS AVANT ALARME LOW LOW LEVEL" %
%   T4:23.PRE  "TEMPS AVANT ALARME LOW LOW LEVEL" %

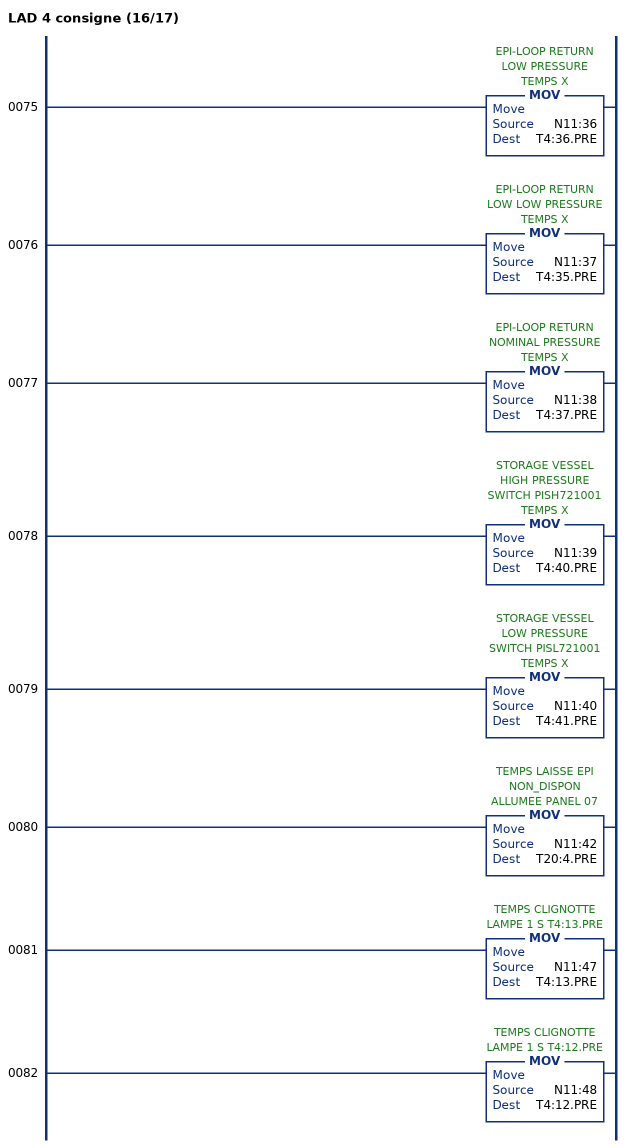
% Rung: 75 %
SOR MOV N11:36 T4:36.PRE EOR
%   N11:36  "EPI-LOOP RETURN LOW PRESSURE TEMPS X" %
%   T4:36.PRE  "EPI-LOOP RETURN LOW PRESSURE TEMPS X" %
% Rung: 76 %
SOR MOV N11:37 T4:35.PRE EOR
%   N11:37  "EPI-LOOP RETURN LOW LOW PRESSURE TEMPS X" %
%   T4:35.PRE  "EPI-LOOP RETURN LOW LOW PRESSURE TEMPS X" %
% Rung: 77 %
SOR MOV N11:38 T4:37.PRE EOR
%   N11:38  "EPI-LOOP RETURN NOMINAL PRESSURE TEMPS X" %
%   T4:37.PRE  "EPI-LOOP RETURN NOMINAL PRESSURE TEMPS X" %
% Rung: 78 %
SOR MOV N11:39 T4:40.PRE EOR
%   N11:39  "STORAGE VESSEL HIGH PRESSURE SWITCH PISH721001 TEMPS X" %
%   T4:40.PRE  "STORAGE VESSEL HIGH PRESSURE SWITCH PISH721001 TEMPS X" %
% Rung: 79 %
SOR MOV N11:40 T4:41.PRE EOR
%   N11:40  "STORAGE VESSEL LOW PRESSURE SWITCH PISL721001 TEMPS X" %
%   T4:41.PRE  "STORAGE VESSEL LOW PRESSURE SWITCH PISL721001 TEMPS X" %
% Rung: 80 %
SOR MOV N11:42 T20:4.PRE EOR
%   N11:42  "TEMPS LAISSE EPI NON_DISPON ALLUMEE PANEL 07" %
%   T20:4.PRE  "TEMPS LAISSE EPI NON_DISPON ALLUMEE PANEL 07" %
% Rung: 81 %
SOR MOV N11:47 T4:13.PRE EOR
%   N11:47  "TEMPS CLIGNOTTE LAMPE 1S" %
%   T4:13.PRE  "TEMPS CLIGNOTTE LAMPE 1 S T4:13.PRE" %
% Rung: 82 %
SOR MOV N11:48 T4:12.PRE EOR
%   N11:48  "TEMPS CLIGNOTTE LAMPE 1S" %
%   T4:12.PRE  "TEMPS CLIGNOTTE LAMPE 1 S T4:12.PRE" %

